FUNCTION_BLOCK FB_GreenShapeDecorator EXTENDS FB_ShapeDecorator

METHOD FB_init : BOOL
VAR_INPUT
	bInitRetains : BOOL; // if TRUE, the retain variables are initialized (warm start / cold start)
	bInCopyCode : BOOL;  // if TRUE, the instance afterwards gets moved into the copy code (online change)
	iDecoratedShape : I_Shape;
END_VAR
SUPER^._iDecoratedShape := iDecoratedShape;
END_METHOD


METHOD  M_Draw : BOOL
M_Draw := SUPER^._iDecoratedShape.M_Draw();
M_SetGreenBorder(SUPER^._iDecoratedShape);
END_METHOD

METHOD PRIVATE M_SetGreenBorder
VAR_INPUT
	iDecoratedShape : I_Shape;
END_VAR
ADSLOGSTR(ADSLOG_MSGTYPE_HINT, 'Border Color : Green', '');
END_METHOD

END_FUNCTION_BLOCK

(* stored: Version 1.1.0.1, ProductVersion 3.1.4024.12
   POU FB_GreenShapeDecorator: Id {8abeb9b3-ec91-4cf7-8b94-e5b7769828bf}, SpecialFunc None
   Method FB_init: Id {20565dae-26ed-4aaa-af6c-db8ef8b86b3c}
   Method M_Draw: Id {62b890bb-b0ca-4b36-8611-51ce89e030da}
   Method M_SetGreenBorder: Id {2703fbca-b3cd-46af-a0e5-31f446bc0af8} *)
